{attribute addProperty BoxType "EP6002-0002-0023"}
{attribute addProperty Id "COM_TxPDO_Map_Inputs_ChannelAT %I*ARRAY[0..1] OF COM_TxPDO_Map_Inputs_Channel_18212A5E384480COM_RxPDO_Map_Outputs_ChannelAT %Q*ARRAY[0..1] OF COM_RxPDO_Map_Outputs_Channel_F536B385384480WcStateAT %I*WcState_98A4DF7520.250InfoDataAT %I*InfoData_BC63D37F80100"}
{attribute addProperty CRC "314694980"}
{attribute addProperty SizeInBites "850"}
{attribute addProperty SizeInBytes "106.25"}
TYPE EP6002_FC20A988 :
STRUCT
	{attribute addProperty Name "COM_TxPDO_Map_Inputs_Channel"}
	COM_TxPDO_Map_Inputs_Channel : ARRAY[0..1] OF COM_TxPDO_Map_Inputs_Channel_18212A5E;
	{attribute addProperty Name "COM_RxPDO_Map_Outputs_Channel"}
	COM_RxPDO_Map_Outputs_Channel : ARRAY[0..1] OF COM_RxPDO_Map_Outputs_Channel_F536B385;
	{attribute addProperty Name "WcState"}
	WcState : WcState_98A4DF75;
	{attribute addProperty Name "InfoData"}
	InfoData : InfoData_BC63D37F;
END_STRUCT
END_TYPE

(* stored: Version 1.2.0.0, ProductVersion 3.1.4024.9
   DUT EP6002_FC20A988: Id {ae678952-a68c-45ae-ade7-1cb7ed4f1640} *)
